// TIA Portal V16 export
// export: Created 2024-06-24T15:42:27.2875043Z, ExportSetting WithDefaults, DisplayName Totally Integrated Automation Portal, DisplayVersion V16, DisplayName TIA Portal Version Control Interface, DisplayVersion V16, DisplayName TIA Portal Openness, DisplayVersion V16, DisplayName STEP 7 Professional, DisplayVersion V16, DisplayName STEP 7 Safety, DisplayVersion V16, DisplayName WinCC Advanced, DisplayVersion V16
ORGANIZATION_BLOCK "OB_Encoder"   // OB123, LAD, ProgramCycle
TITLE = "Main Program Sweep (Cycle)"
{ S7_Optimized_Access := 'TRUE' }
VERSION : 0.1
// stored: AutoNumber true, IsIECCheckEnabled false, SetENOAutomatically false
   VAR_INPUT
      Initial_Call : Bool;   // Initial call of this OB
      Remanence : Bool;   // =True, if remanent data are available
   END_VAR
   VAR_TEMP   // added for the SCL form of the ladder/FBD networks
      _w1 : Bool;
      _w2 : Bool;
   END_VAR
BEGIN

REGION Network 1
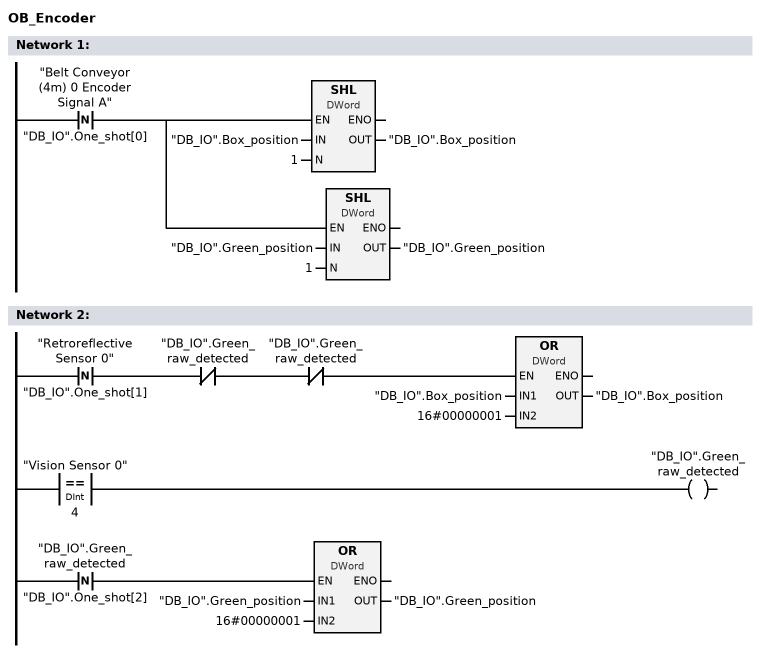
   RUNG wire#powerrail
      N_Contact(operand := "Belt Conveyor (4m) 0 Encoder Signal A", bit := "DB_IO".One_shot[0])
      wire#w1
      { S7_Templates := "SrcType := DWord" } Shl(in := "DB_IO".Box_position, n := 1, out => "DB_IO".Box_position)
   END_RUNG
   RUNG wire#w1
      { S7_Templates := "SrcType := DWord" } Shl(in := "DB_IO".Green_position, n := 1, out => "DB_IO".Green_position)
   END_RUNG
   // the same network as SCL:
   #_w1 := NOT "Belt Conveyor (4m) 0 Encoder Signal A" AND "DB_IO".One_shot[0];   // falling edge of "Belt Conveyor (4m) 0 Encoder Signal A"
   "DB_IO".One_shot[0] := "Belt Conveyor (4m) 0 Encoder Signal A";
   IF #_w1 THEN
       "DB_IO".Box_position := SHL(IN := "DB_IO".Box_position, N := 1);
       "DB_IO".Green_position := SHL(IN := "DB_IO".Green_position, N := 1);
   END_IF;
END_REGION

REGION Network 2
   #_w1 := NOT "Retroreflective Sensor 0" AND "DB_IO".One_shot[1];   // falling edge of "Retroreflective Sensor 0"
   "DB_IO".One_shot[1] := "Retroreflective Sensor 0";
   IF #_w1 AND NOT "DB_IO".Green_raw_detected AND NOT "DB_IO".Green_raw_detected THEN
       "DB_IO".Box_position := "DB_IO".Box_position OR 16#00000001;
   END_IF;
   "DB_IO".Green_raw_detected := "Vision Sensor 0" = 4;
   #_w2 := NOT "DB_IO".Green_raw_detected AND "DB_IO".One_shot[2];   // falling edge of "DB_IO".Green_raw_detected
   "DB_IO".One_shot[2] := "DB_IO".Green_raw_detected;
   IF #_w2 THEN "DB_IO".Green_position := "DB_IO".Green_position OR 16#00000001; END_IF;
END_REGION
END_ORGANIZATION_BLOCK
